(* Logix 5000 project; controller exercice vendor 1 type 14 code 150 rev 37.11; software revision 37.00 *)

TASK MainTask (continuous, watchdog 500 ms) : MainProgram

MODULES
   Local : vendor 1 type 14 code 150 (Compact 0, rev 37.11)
      Discrete_IO : Embedded (Compact 1, rev 3.1, Output RPI 20 ms)
      Analog_IO : Embedded (Compact 2, rev 1.1, Output RPI 80 ms)
      Counters : Embedded (Compact 3, rev 1.1, Output RPI 20 ms)
END_MODULES

VAR_GLOBAL   (* controller tags *)
   M1 : ALIAS FOR Local:1:O.Data.0;
   START1 : ALIAS FOR Local:1:I.Data.11;
   START2 : ALIAS FOR Local:1:I.Data.8;
   STOP : ALIAS FOR Local:1:I.Data.12;
   STOP1 : ALIAS FOR Local:1:I.Data.9;
END_VAR

PROGRAM MainProgram   (* main routine MainRoutine *)

ROUTINE MainRoutine   (* ladder *)
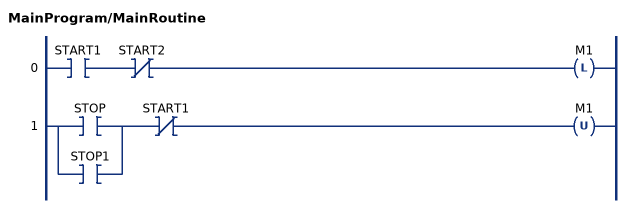
   0: XIC(START1)XIO(START2)OTL(M1);
   1: [XIC(STOP) ,XIC(STOP1) ]XIO(START1)OTU(M1);
END_ROUTINE
END_PROGRAM
